// TIA Portal V20 export
DATA_BLOCK "PM06"   // DB335
// stored: MemoryReserve 100
   VAR
      "CATHODE GLASS CLEANING ON" : Bool := FALSE;
      SPARE : Bool := FALSE;
      "CATHODE MAIN NG P&P UP" : Bool := FALSE;
      "CATHODE MAIN NG P&P DOWN" : Bool := FALSE;
      "CATHODE MAIN NG P&P 1st FORWARD" : Bool := FALSE;
      "CATHODE MAIN NG P&P 1st BACKWARD" : Bool := FALSE;
      "CATHODE MAIN NG P&P 2nd FORWARD" : Bool := FALSE;
      "CATHODE MAIN NG P&P 2nd BACKWARD" : Bool := FALSE;
      "CATHODE FIX FRONT&REAR FORWARD" : Bool := FALSE;
      "CATHODE FIX FRONT&REAR BACKWARD" : Bool := FALSE;
      "CATHODE MAIN P&P#1 Rotary CW" : Bool := FALSE;
      "CATHODE MAIN P&P#1 Rotary CCW" : Bool := FALSE;
      "CATHODE NG BOX LIFT UP" : Bool := FALSE;
      "CATHODE NG BOX LIFT DOWN" : Bool := FALSE;
      "CATHODE NG BOX LOCK UP" : Bool := FALSE;
      "CATHODE NG BOX LOCK DOWN" : Bool := FALSE;
   END_VAR
BEGIN
END_DATA_BLOCK
